% RSLogix 500 project pump_project.RSS, saved by version 8.30.00.16 %
PROJECT "UNTITLED"    % processor: Bul.1763 MicroLogix 1100 Series B %

PROGRAM FILES
  LAD 2 "MAIN"  4 rungs
  LAD 3 "INPUT"  4 rungs  % input and output signals %
  LAD 4 "CONTROL"  7 rungs  % pump control logic %
  LAD 5 "OUTPUT"  3 rungs  % output signals %

DATA FILES
  O0 OUTPUT  6 elements
  I1 INPUT  12 elements
  S2 STATUS  66 elements
  B3 BINARY  1 elements
  T4 TIMER  2 elements
  C5 COUNTER  1 elements
  R6 CONTROL  1 elements
  N7 INTEGER  1 elements
  F8 FLOAT  1 elements

LADDER 2 "MAIN"
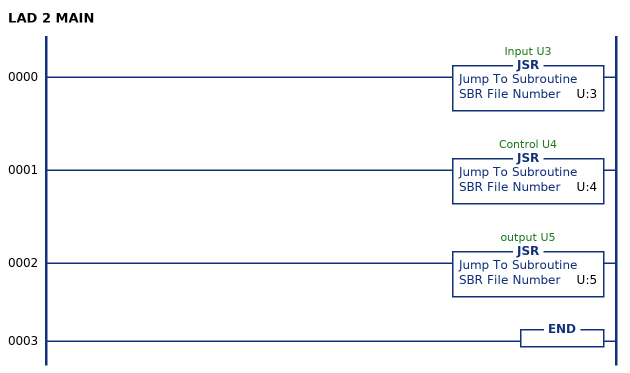
% Rung: 0 %
SOR JSR U:3 EOR
%   U:3  U3  "Input" %
% Rung: 1 %
SOR JSR U:4 EOR
%   U:4  U4  "Control" %
% Rung: 2 %
SOR JSR U:5 EOR
%   U:5  U5  "output" %
% Rung: 3 %
SOR END EOR

LADDER 3 "INPUT"    % input and output signals %
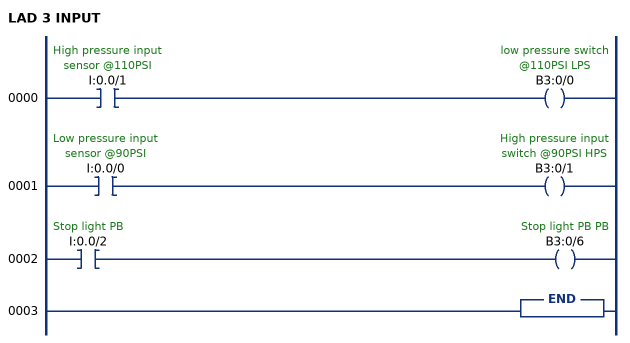
% Rung: 0 %
SOR XIC I:0.0/1 OTE B3:0/0 EOR
%   I:0.0/1  "High pressure input sensor @110PSI" %
%   B3:0/0  LPS  "low pressure switch @110PSI" %
% Rung: 1 %
SOR XIC I:0.0/0 OTE B3:0/1 EOR
%   I:0.0/0  "Low pressure input sensor @90PSI" %
%   B3:0/1  HPS  "High pressure input switch @90PSI" %
% Rung: 2 %
SOR XIC I:0.0/2 OTE B3:0/6 EOR
%   I:0.0/2  "Stop light PB" %
%   B3:0/6  PB  "Stop light PB" %
% Rung: 3 %
SOR END EOR

LADDER 4 "CONTROL"    % pump control logic %
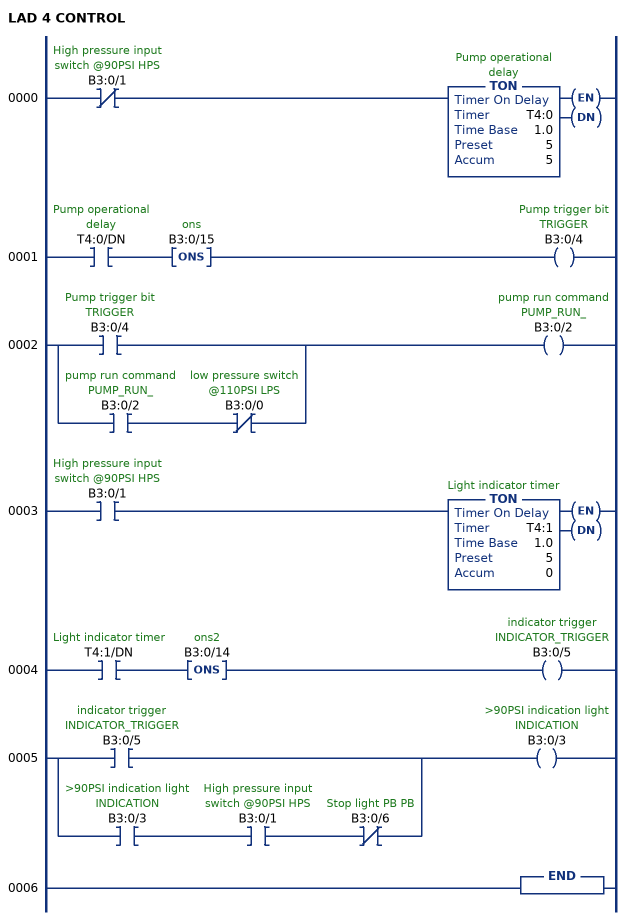
% Rung: 0 %
SOR XIO B3:0/1 TON T4:0 1.0 5 5 EOR
%   B3:0/1  HPS  "High pressure input switch @90PSI" %
%   T4:0  "Pump operational delay" %
% Rung: 1 %
SOR XIC T4:0/DN ONS B3:0/15 OTE B3:0/4 EOR
%   T4:0  "Pump operational delay" %
%   B3:0/15  "ons" %
%   B3:0/4  TRIGGER  "Pump trigger bit" %
% Rung: 2 %
SOR BST XIC B3:0/4 NXB XIC B3:0/2 XIO B3:0/0 BND OTE B3:0/2 EOR
%   B3:0/4  TRIGGER  "Pump trigger bit" %
%   B3:0/2  PUMP_RUN_  "pump run command" %
%   B3:0/0  LPS  "low pressure switch @110PSI" %
% Rung: 3 %
SOR XIC B3:0/1 TON T4:1 1.0 5 0 EOR
%   B3:0/1  HPS  "High pressure input switch @90PSI" %
%   T4:1  "Light indicator timer" %
% Rung: 4 %
SOR XIC T4:1/DN ONS B3:0/14 OTE B3:0/5 EOR
%   T4:1  "Light indicator timer" %
%   B3:0/14  "ons2" %
%   B3:0/5  INDICATOR_TRIGGER  "indicator trigger" %
% Rung: 5 %
SOR BST XIC B3:0/5 NXB XIC B3:0/3 XIC B3:0/1 XIO B3:0/6 BND OTE B3:0/3 EOR
%   B3:0/5  INDICATOR_TRIGGER  "indicator trigger" %
%   B3:0/3  INDICATION  ">90PSI indication light" %
%   B3:0/1  HPS  "High pressure input switch @90PSI" %
%   B3:0/6  PB  "Stop light PB" %
% Rung: 6 %
SOR END EOR

LADDER 5 "OUTPUT"    % output signals %
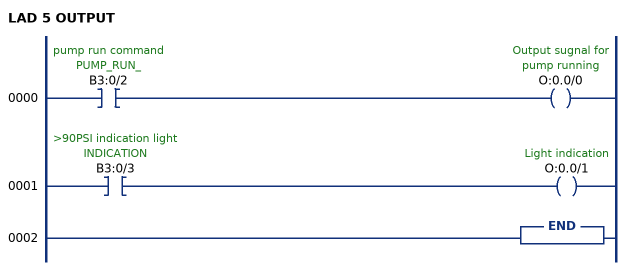
% Rung: 0 %
SOR XIC B3:0/2 OTE O:0.0/0 EOR
%   B3:0/2  PUMP_RUN_  "pump run command" %
%   O:0.0/0  "Output sugnal for pump running" %
% Rung: 1 %
SOR XIC B3:0/3 OTE O:0.0/1 EOR
%   B3:0/3  INDICATION  ">90PSI indication light" %
%   O:0.0/1  "Light indication" %
% Rung: 2 %
SOR END EOR

OTHER DOCUMENTED ADDRESSES
  B3:0/13  "ons3"
  T4:0/0  "Pump operational delay"

DATA TABLE (non-zero values as saved)
DATA B3
% B3:0 % 0X8004
DATA T4
% .PRE .ACC %
% T4:0 % 5 5
% T4:1 % 5 0
